TYPE ACRMemoryStringEvent EXTENDS ACRMemoryEvent :
STRUCT
	_Value : STRING(255);
END_STRUCT
END_TYPE

(* stored: Version 1.1.0.1, ProductVersion 3.1.4020.12
   DUT ACRMemoryStringEvent: Id {cd25e492-a905-4e83-9b18-0c097e51dffb} *)
